VAR_GLOBAL CONSTANT
    TcUnit_ResultExportXmlPath : T_MaxString :=
        'C:\TwinCAT\3.1\Boot\Plc\TcUnitResults.xml';
END_VAR

(* stored: Version 1.1.0.1
   GVL GVL_TcUnit: Id {60c03689-e94f-4d80-8caf-13eb6f341046} *)
